% RSLogix 500 project Evaluacion.RSS, saved by version 8.40.00.08 %
PROJECT "UNTITLED"    % processor: MicroLogix 1200 %

PROGRAM FILES
  LAD 2 "MAIN"  4 rungs
  LAD 3 "ENTRADAS"  7 rungs
  LAD 4 "SALIDAS"  8 rungs
  LAD 6 "AUTOMATICO"  18 rungs
  LAD 7 "PARPADEOS"  5 rungs

DATA FILES
  O0 OUTPUT  4 elements
  I1 INPUT  4 elements
  S2 STATUS  66 elements
  B3 BINARY  2 elements
  T4 TIMER  5 elements
  C5 COUNTER  2 elements
  R6 CONTROL  1 elements
  N7 INTEGER  1 elements
  F8 FLOAT  1 elements
  B30   1 elements

LADDER 2 "MAIN"
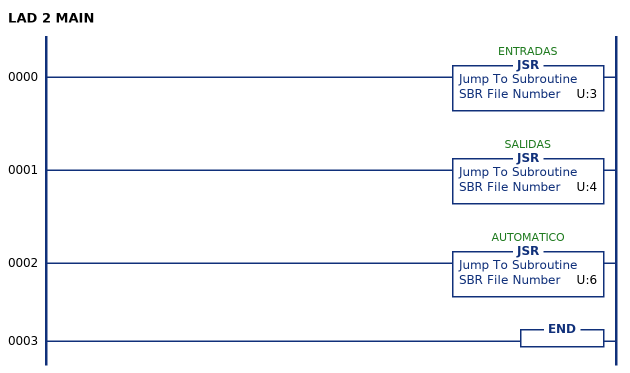
% Rung: 0 %
SOR JSR U:3 EOR
%   U:3  ENTRADAS %
% Rung: 1 %
SOR JSR U:4 EOR
%   U:4  SALIDAS %
% Rung: 2 %
SOR JSR U:6 EOR
%   U:6  AUTOMATICO %
% Rung: 3 %
SOR END EOR

LADDER 3 "ENTRADAS"
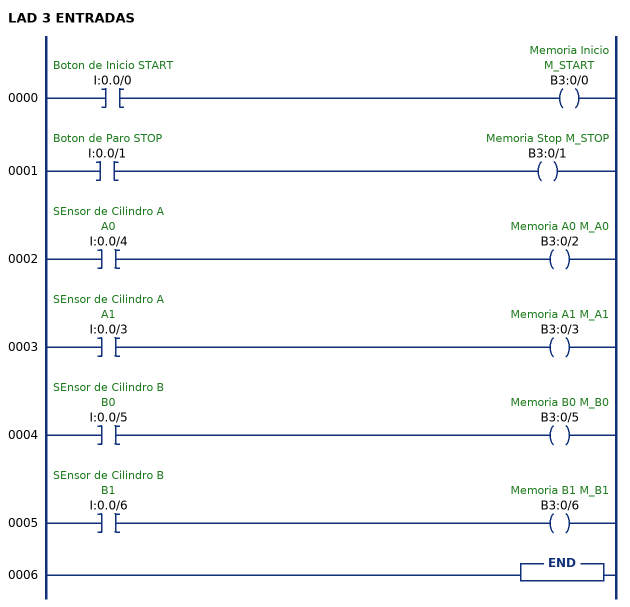
% Rung: 0 %
SOR XIC I:0.0/0 OTE B3:0/0 EOR
%   I:0.0/0  START  "Boton de Inicio" %
%   B3:0/0  M_START  "Memoria Inicio" %
% Rung: 1 %
SOR XIC I:0.0/1 OTE B3:0/1 EOR
%   I:0.0/1  STOP  "Boton de Paro" %
%   B3:0/1  M_STOP  "Memoria Stop" %
% Rung: 2 %
SOR XIC I:0.0/4 OTE B3:0/2 EOR
%   I:0.0/4  A0  "SEnsor de Cilindro A" %
%   B3:0/2  M_A0  "Memoria A0" %
% Rung: 3 %
SOR XIC I:0.0/3 OTE B3:0/3 EOR
%   I:0.0/3  A1  "SEnsor de Cilindro A" %
%   B3:0/3  M_A1  "Memoria A1" %
% Rung: 4 %
SOR XIC I:0.0/5 OTE B3:0/5 EOR
%   I:0.0/5  B0  "SEnsor de Cilindro B" %
%   B3:0/5  M_B0  "Memoria B0" %
% Rung: 5 %
SOR XIC I:0.0/6 OTE B3:0/6 EOR
%   I:0.0/6  B1  "SEnsor de Cilindro B" %
%   B3:0/6  M_B1  "Memoria B1" %
% Rung: 6 %
SOR END EOR

LADDER 4 "SALIDAS"
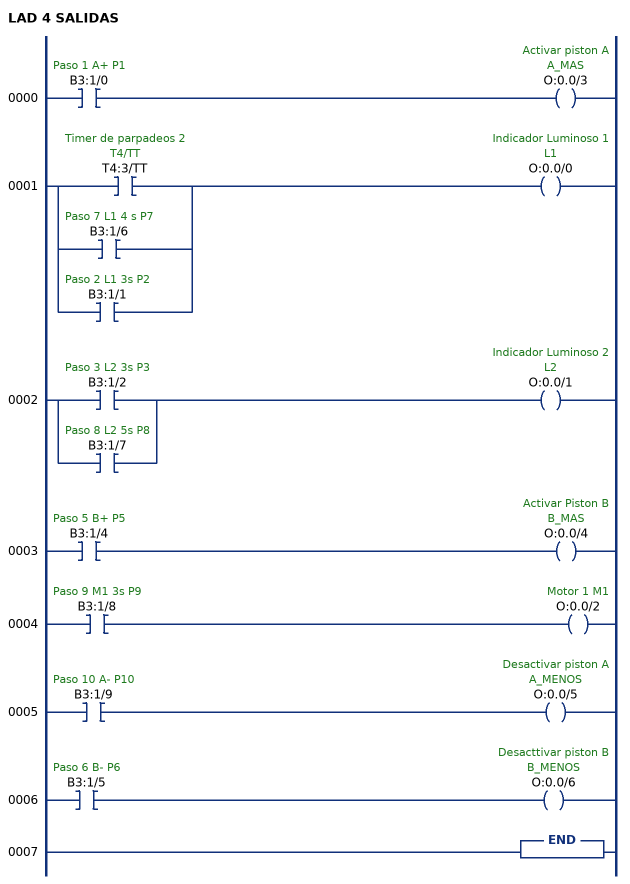
% Rung: 0 %
SOR XIC B3:1/0 OTE O:0.0/3 EOR
%   B3:1/0  P1  "Paso 1 A+" %
%   O:0.0/3  A_MAS  "Activar piston A" %
% Rung: 1 %
SOR BST XIC T4:3/TT NXB XIC B3:1/6 NXB XIC B3:1/1 BND OTE O:0.0/0 EOR
%   T4:3  T4  "Timer de parpadeos 2" %
%   B3:1/6  P7  "Paso 7 L1 4 s" %
%   B3:1/1  P2  "Paso 2 L1 3s" %
%   O:0.0/0  L1  "Indicador Luminoso 1" %
% Rung: 2 %
SOR BST XIC B3:1/2 NXB XIC B3:1/7 BND OTE O:0.0/1 EOR
%   B3:1/2  P3  "Paso 3 L2 3s" %
%   B3:1/7  P8  "Paso 8 L2 5s" %
%   O:0.0/1  L2  "Indicador Luminoso 2" %
% Rung: 3 %
SOR XIC B3:1/4 OTE O:0.0/4 EOR
%   B3:1/4  P5  "Paso 5 B+" %
%   O:0.0/4  B_MAS  "Activar Piston B" %
% Rung: 4 %
SOR XIC B3:1/8 OTE O:0.0/2 EOR
%   B3:1/8  P9  "Paso 9 M1 3s" %
%   O:0.0/2  M1  "Motor 1" %
% Rung: 5 %
SOR XIC B3:1/9 OTE O:0.0/5 EOR
%   B3:1/9  P10  "Paso 10 A-" %
%   O:0.0/5  A_MENOS  "Desactivar piston A" %
% Rung: 6 %
SOR XIC B3:1/5 OTE O:0.0/6 EOR
%   B3:1/5  P6  "Paso 6 B-" %
%   O:0.0/6  B_MENOS  "Desacttivar piston B" %
% Rung: 7 %
SOR END EOR

LADDER 6 "AUTOMATICO"
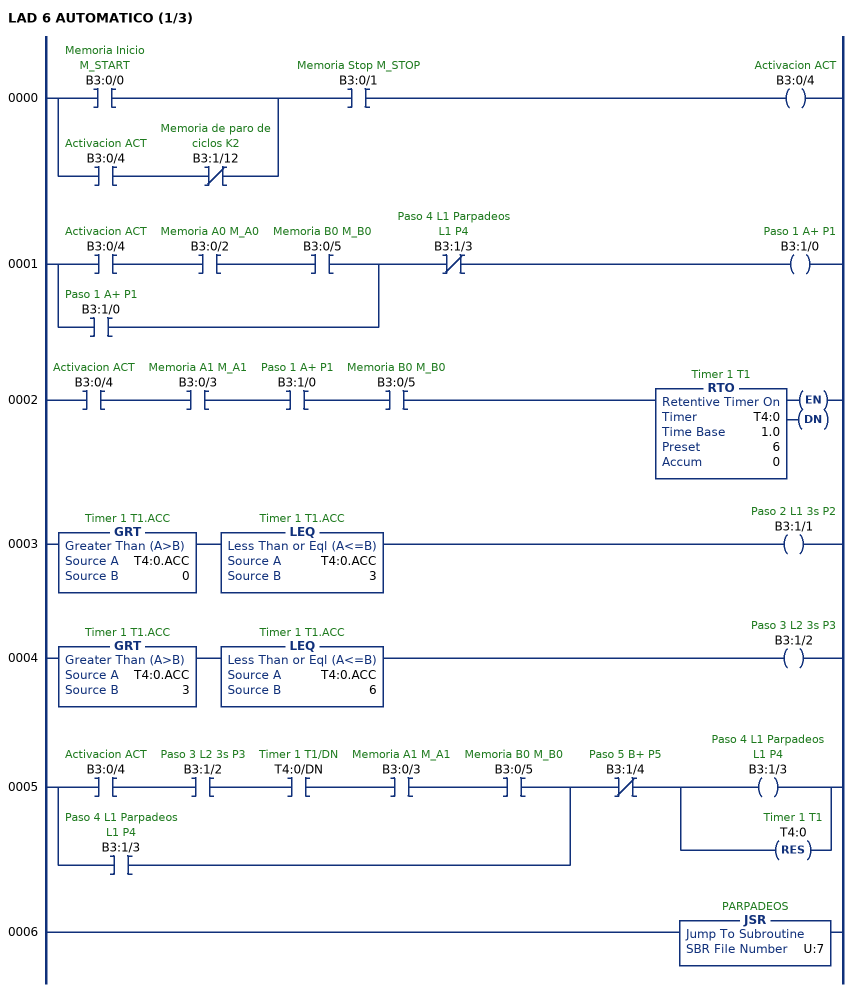
% Rung: 0 %
SOR BST XIC B3:0/0 NXB XIC B3:0/4 XIO B3:1/12 BND XIC B3:0/1 OTE B3:0/4 EOR
%   B3:0/0  M_START  "Memoria Inicio" %
%   B3:0/4  ACT  "Activacion" %
%   B3:1/12  K2  "Memoria de paro de ciclos" %
%   B3:0/1  M_STOP  "Memoria Stop" %
% Rung: 1 %
SOR BST XIC B3:0/4 XIC B3:0/2 XIC B3:0/5 NXB XIC B3:1/0 BND XIO B3:1/3 OTE B3:1/0 EOR
%   B3:0/4  ACT  "Activacion" %
%   B3:0/2  M_A0  "Memoria A0" %
%   B3:0/5  M_B0  "Memoria B0" %
%   B3:1/0  P1  "Paso 1 A+" %
%   B3:1/3  P4  "Paso 4 L1 Parpadeos L1" %
% Rung: 2 %
SOR XIC B3:0/4 XIC B3:0/3 XIC B3:1/0 XIC B3:0/5 RTO T4:0 1.0 6 0 EOR
%   B3:0/4  ACT  "Activacion" %
%   B3:0/3  M_A1  "Memoria A1" %
%   B3:1/0  P1  "Paso 1 A+" %
%   B3:0/5  M_B0  "Memoria B0" %
%   T4:0  T1  "Timer 1" %
% Rung: 3 %
SOR GRT T4:0.ACC 0 LEQ T4:0.ACC 3 OTE B3:1/1 EOR
%   T4:0  T1  "Timer 1" %
%   B3:1/1  P2  "Paso 2 L1 3s" %
% Rung: 4 %
SOR GRT T4:0.ACC 3 LEQ T4:0.ACC 6 OTE B3:1/2 EOR
%   T4:0  T1  "Timer 1" %
%   B3:1/2  P3  "Paso 3 L2 3s" %
% Rung: 5 %
SOR BST XIC B3:0/4 XIC B3:1/2 XIC T4:0/DN XIC B3:0/3 XIC B3:0/5 NXB XIC B3:1/3 BND XIO B3:1/4 BST OTE B3:1/3 NXB RES T4:0 BND EOR
%   B3:0/4  ACT  "Activacion" %
%   B3:1/2  P3  "Paso 3 L2 3s" %
%   T4:0  T1  "Timer 1" %
%   B3:0/3  M_A1  "Memoria A1" %
%   B3:0/5  M_B0  "Memoria B0" %
%   B3:1/3  P4  "Paso 4 L1 Parpadeos L1" %
%   B3:1/4  P5  "Paso 5 B+" %
% Rung: 6 %
SOR JSR U:7 EOR
%   U:7  PARPADEOS %

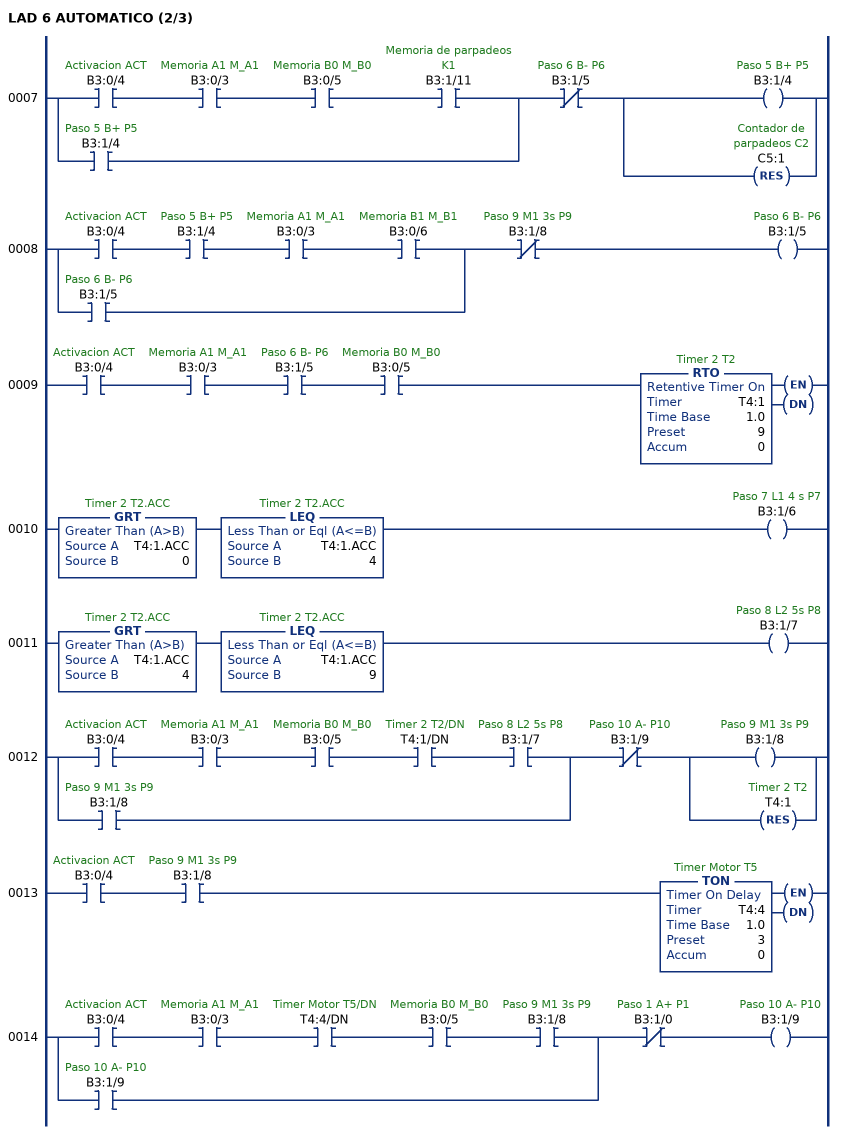
% Rung: 7 %
SOR BST XIC B3:0/4 XIC B3:0/3 XIC B3:0/5 XIC B3:1/11 NXB XIC B3:1/4 BND XIO B3:1/5 BST OTE B3:1/4 NXB RES C5:1 BND EOR
%   B3:0/4  ACT  "Activacion" %
%   B3:0/3  M_A1  "Memoria A1" %
%   B3:0/5  M_B0  "Memoria B0" %
%   B3:1/11  K1  "Memoria de parpadeos" %
%   B3:1/4  P5  "Paso 5 B+" %
%   B3:1/5  P6  "Paso 6 B-" %
%   C5:1  C2  "Contador de parpadeos" %
% Rung: 8 %
SOR BST XIC B3:0/4 XIC B3:1/4 XIC B3:0/3 XIC B3:0/6 NXB XIC B3:1/5 BND XIO B3:1/8 OTE B3:1/5 EOR
%   B3:0/4  ACT  "Activacion" %
%   B3:1/4  P5  "Paso 5 B+" %
%   B3:0/3  M_A1  "Memoria A1" %
%   B3:0/6  M_B1  "Memoria B1" %
%   B3:1/5  P6  "Paso 6 B-" %
%   B3:1/8  P9  "Paso 9 M1 3s" %
% Rung: 9 %
SOR XIC B3:0/4 XIC B3:0/3 XIC B3:1/5 XIC B3:0/5 RTO T4:1 1.0 9 0 EOR
%   B3:0/4  ACT  "Activacion" %
%   B3:0/3  M_A1  "Memoria A1" %
%   B3:1/5  P6  "Paso 6 B-" %
%   B3:0/5  M_B0  "Memoria B0" %
%   T4:1  T2  "Timer 2" %
% Rung: 10 %
SOR GRT T4:1.ACC 0 LEQ T4:1.ACC 4 OTE B3:1/6 EOR
%   T4:1  T2  "Timer 2" %
%   B3:1/6  P7  "Paso 7 L1 4 s" %
% Rung: 11 %
SOR GRT T4:1.ACC 4 LEQ T4:1.ACC 9 OTE B3:1/7 EOR
%   T4:1  T2  "Timer 2" %
%   B3:1/7  P8  "Paso 8 L2 5s" %
% Rung: 12 %
SOR BST XIC B3:0/4 XIC B3:0/3 XIC B3:0/5 XIC T4:1/DN XIC B3:1/7 NXB XIC B3:1/8 BND XIO B3:1/9 BST OTE B3:1/8 NXB RES T4:1 BND EOR
%   B3:0/4  ACT  "Activacion" %
%   B3:0/3  M_A1  "Memoria A1" %
%   B3:0/5  M_B0  "Memoria B0" %
%   T4:1  T2  "Timer 2" %
%   B3:1/7  P8  "Paso 8 L2 5s" %
%   B3:1/8  P9  "Paso 9 M1 3s" %
%   B3:1/9  P10  "Paso 10 A-" %
% Rung: 13 %
SOR XIC B3:0/4 XIC B3:1/8 TON T4:4 1.0 3 0 EOR
%   B3:0/4  ACT  "Activacion" %
%   B3:1/8  P9  "Paso 9 M1 3s" %
%   T4:4  T5  "Timer Motor" %
% Rung: 14 %
SOR BST XIC B3:0/4 XIC B3:0/3 XIC T4:4/DN XIC B3:0/5 XIC B3:1/8 NXB XIC B3:1/9 BND XIO B3:1/0 OTE B3:1/9 EOR
%   B3:0/4  ACT  "Activacion" %
%   B3:0/3  M_A1  "Memoria A1" %
%   T4:4  T5  "Timer Motor" %
%   B3:0/5  M_B0  "Memoria B0" %
%   B3:1/8  P9  "Paso 9 M1 3s" %
%   B3:1/9  P10  "Paso 10 A-" %
%   B3:1/0  P1  "Paso 1 A+" %

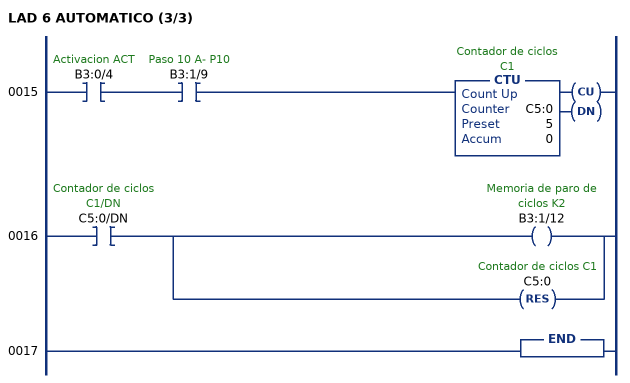
% Rung: 15 %
SOR XIC B3:0/4 XIC B3:1/9 CTU C5:0 5 0 EOR
%   B3:0/4  ACT  "Activacion" %
%   B3:1/9  P10  "Paso 10 A-" %
%   C5:0  C1  "Contador de ciclos" %
% Rung: 16 %
SOR XIC C5:0/DN BST OTE B3:1/12 NXB RES C5:0 BND EOR
%   C5:0  C1  "Contador de ciclos" %
%   B3:1/12  K2  "Memoria de paro de ciclos" %
% Rung: 17 %
SOR END EOR

LADDER 7 "PARPADEOS"
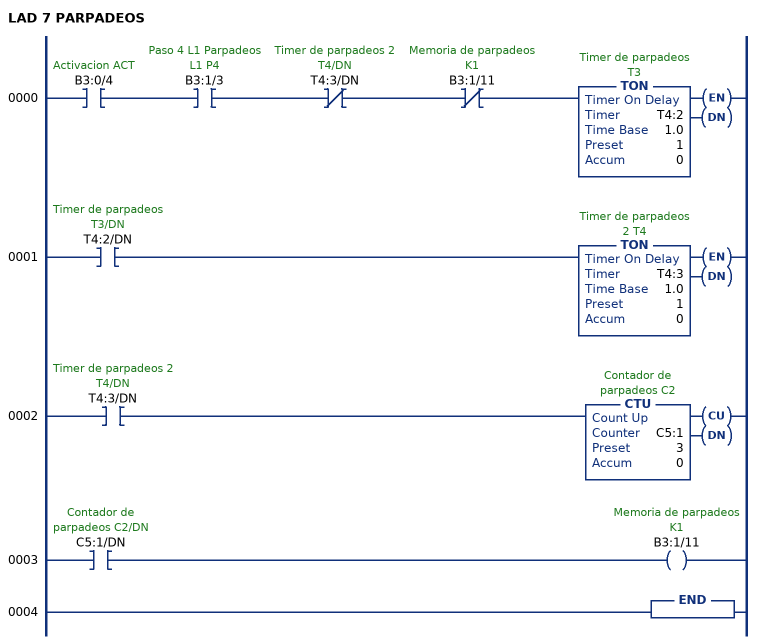
% Rung: 0 %
SOR XIC B3:0/4 XIC B3:1/3 XIO T4:3/DN XIO B3:1/11 TON T4:2 1.0 1 0 EOR
%   B3:0/4  ACT  "Activacion" %
%   B3:1/3  P4  "Paso 4 L1 Parpadeos L1" %
%   T4:3  T4  "Timer de parpadeos 2" %
%   B3:1/11  K1  "Memoria de parpadeos" %
%   T4:2  T3  "Timer de parpadeos" %
% Rung: 1 %
SOR XIC T4:2/DN TON T4:3 1.0 1 0 EOR
%   T4:2  T3  "Timer de parpadeos" %
%   T4:3  T4  "Timer de parpadeos 2" %
% Rung: 2 %
SOR XIC T4:3/DN CTU C5:1 3 0 EOR
%   T4:3  T4  "Timer de parpadeos 2" %
%   C5:1  C2  "Contador de parpadeos" %
% Rung: 3 %
SOR XIC C5:1/DN OTE B3:1/11 EOR
%   C5:1  C2  "Contador de parpadeos" %
%   B3:1/11  K1  "Memoria de parpadeos" %
% Rung: 4 %
SOR END EOR

OTHER DOCUMENTED ADDRESSES
  B3:1/10  PA  "Paso Auxiliar"

DATA TABLE (non-zero values as saved)
DATA B3
% B3:0 % 0X0026 0X0000
DATA T4
% .PRE .ACC %
% T4:0 % 6 0
% T4:1 % 9 0
% T4:2 % 1 0
% T4:3 % 1 0
% T4:4 % 3 0
DATA C5
% .PRE .ACC %
% C5:0 % 5 0
% C5:1 % 3 0
